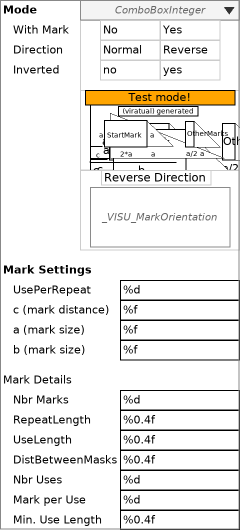
VISUALIZATION _VISU_MarkModes  // 240x530
VAR_IN_OUT
  mInst : FB_MarkCamera_WEU;
END_VAR
    Rectangle (80,20 160x80)
    Rectangle (80,90 160x80)
    Rectangle (0,0 120x20), "Mode"
    Rectangle (120,300 120x20), "%f", text variable: mInst.fMarkSpec_c
        OnMouseClick: write the text variable via Default
    Rectangle (120,280 120x20), "%d", text variable: mInst.nUsePerRepeat
        OnMouseClick: write the text variable via Default
    Rectangle (10,280 110x20), "UsePerRepeat"
    Rectangle (10,320 110x20), "a (mark size)", input disabled if: TRUE
    Rectangle (10,300 110x20), "c (mark distance)", input disabled if: TRUE
    Rectangle (120,320 120x20), "%f", text variable: mInst.fMarkSpec_a, colour toggle: mInst.fMarkSpec_a = 0
        OnMouseClick: write the text variable via Default
    ComboBoxInteger (80,0 160x20), variable: mInst.eMarkMode, text list: 'TL_MarkMode'
    Rectangle (10,340 110x20), "b (mark size)", input disabled if: TRUE
    Rectangle (120,340 120x20), "%f", text variable: mInst.fMarkSpec_b
        OnMouseClick: write the text variable via Default
    Group (90,95 147x63), invisible if: mInst.eMarkMode <> E_MarkMode.AutoDefault
        Polyline (0,0) (0,84) (121,84)
        Polygon (79,28) (79,65) (117,65)
        Rectangle (19,28 60x37)
        Rectangle (37,64 26x19), "2*a"
        Rectangle (81,64 37x19), "a"
        Rectangle (9,37 26x19), "a"
        Rectangle (19,37 61x19), "StartMark"
        Line (1,64) (17,64)
        Rectangle (4,65 26x19), "c"
        Rectangle (79,37 26x19), "a"
        Group (129,28 76x55)
            Rectangle (3,0 13x37)
            Polygon (16,0) (16,37) (53,37)
            Rectangle (0,36 26x19), "a/2"
            Rectangle (1,9 75x19), "OtherMarks"
            Rectangle (20,36 37x19), "a"
    Group (90,95 113x65), invisible if: mInst.eMarkMode <> E_MarkMode.OneDefault
        Polyline (0,0) (0,103) (147,103)
        Polygon (95,33) (95,78) (141,78)
        Rectangle (23,34 73x45)
        Rectangle (45,78 32x23), "2*a"
        Rectangle (97,78 45x23), "a"
        Rectangle (10,44 32x23), "a"
        Rectangle (23,44 75x23), "StartMark"
        Line (1,78) (21,78)
        Rectangle (0,78 32x23), "c"
        Rectangle (96,44 32x23), "a"
    Group (90,95 100x60), invisible if: mInst.eMarkMode <> E_MarkMode.OneTriangle
        Polyline (0,0) (0,89) (146,89)
        Polygon (20,18) (20,63) (134,63)
        Rectangle (45,64 33x23), "b"
        Rectangle (11,36 33x23), "a"
        Rectangle (23,36 76x23), "StartMark"
        Line (0,63) (19,63)
        Rectangle (0,64 33x23), "c"
    RoundedRectangle (100,40 60x20), "Normal", colour toggle: NOT mInst.bPrintDirReverse
    Rectangle (10,40 110x20), "Direction"
    RoundedRectangle (160,40 60x20), "Reverse", colour toggle: mInst.bPrintDirReverse
    Rectangle (10,20 110x20), "With Mark"
    RoundedRectangle (100,20 60x20), "No", colour toggle: NOT mInst.bPrintMarkExist
    RoundedRectangle (160,20 60x20), "Yes", colour toggle: mInst.bPrintMarkExist
    Rectangle (10,60 110x20), "Inverted", tooltip "Mark is flipped/inverted"
    RoundedRectangle (160,60 60x20), "yes", colour toggle: mInst.bMarkInverted
    RoundedRectangle (100,60 60x20), "no", colour toggle: NOT mInst.bMarkInverted
    Rectangle (80,170 160x80)
    RoundedRectangle (85,90 150x15), "Test mode!", invisible if: mInst.eMarkMode = E_MarkMode.AutoDefault OR mInst.eMarkMode = E_MarkMode.None
    Rectangle (0,260 120x20), "Mark Settings"
    Frame (90,187 140x60)
        shows _VISU_MarkOrientation(mInst := mInst)
    RoundedRectangle (101,170 110x15), "Reverse Direction"
        toggle mInst.bPrintDirReverse
    Rectangle (10,410 110x20), "RepeatLength"
    Rectangle (120,410 120x20), "%0.4f", text variable: mInst.fbMarkDefinition._fImageLength, colour toggle: mInst._bImageLengthError, input disabled if: TRUE
    Rectangle (0,370 120x20), "Mark Details"
    Rectangle (10,430 110x20), "UseLength"
    Rectangle (120,430 120x20), "%0.4f", text variable: mInst.fbMarkDefinition._fUseLength, input disabled if: TRUE
    Rectangle (10,450 110x20), "DistBetweenMasks"
    Rectangle (120,450 120x20), "%0.4f", text variable: mInst.fbMarkDefinition._fDistBetweenMarks, input disabled if: TRUE
    Rectangle (10,470 110x20), "Nbr Uses"
    Rectangle (120,470 120x20), "%d", text variable: mInst.fbMarkDefinition._nUses, input disabled if: TRUE
    Rectangle (10,490 110x20), "Mark per Use"
    Rectangle (120,490 120x20), "%d", text variable: mInst.fbMarkDefinition._nMarksPerUse, input disabled if: TRUE
    Rectangle (10,390 110x20), "Nbr Marks"
    Rectangle (120,390 120x20), "%d", tooltip "teached marks", text variable: mInst.fbMarkDefinition._nMarks, colour toggle: mInst.fbMarkDefinition._nMarks = 0, input disabled if: TRUE
    Rectangle (10,510 110x20), "Min. Use Length"
    Rectangle (120,510 120x20), "%0.4f", text variable: mInst.fbMarkDefinition.fC_MinUseLength, input disabled if: TRUE
    Group (90,106 147x56), invisible if: mInst.eMarkMode <> E_MarkMode.None
        Polyline (0,1) (0,56) (86,56)
        Polygon (56,14) (56,40) (83,40)
        Rectangle (14,14 43x27)
        Rectangle (27,41 19x14), "2*a"
        Rectangle (58,41 27x14), "a"
        Rectangle (6,22 19x14), "a"
        Rectangle (14,22 44x14), "StartMark"
        Line (0,40) (12,40)
        Rectangle (3,42 19x14), "c"
        Rectangle (57,22 19x14), "a"
        Rectangle (95,15 9x26)
        Polygon (104,15) (104,41) (130,41)
        Rectangle (93,41 18x13), "a/2"
        Rectangle (94,21 53x13), "OtherMarks"
        Rectangle (107,41 26x13), "a"
        Rectangle (28,0 80x10), "(viratual) generated"
END_VISUALIZATION

(* stored: Version 1.1.0.1, ProductVersion 3.1.4024.11
   Visu _VISU_MarkModes: Id {9feaaacc-32dc-4df6-a9b7-b018448d9d3b} *)
